// TIA Portal V20 export
TYPE "UDT_FuellstandStatus"
   STRUCT
      IST_AKTUELL : Real;
      IST_GLATT : Real;
      VISU_FABRE : Int;
      Bit8 : Bool;
      Bit9 : Bool;
      Belegt : Bool;
      Bit11 : Bool;
      Bit12 : Bool;
      Bit13 : Bool;
      Bit14 : Bool;
      Bit15 : Bool;
      EINSCHALT : Bool;
      AUSSCHALT : Bool;
      Bit3 : Bool;
      Bit4 : Bool;
      MESS_DB_STOE : Bool;
      SIM_AKTIV : Bool;
      STOE : Bool;
      STOE_NEU : Bool;
   END_STRUCT;
END_TYPE
